FUNCTION_BLOCK ATM_SUB (* Subtracts two TIME values via ATM adapters (F_SUB is ANY_MAGNITUDE, works directly on TIME) *)
  (* Standard: 61499-2; Description: Copyright (c) 2026 HR Agrartechnik GmbH This program and the accompanying materials are made available under the terms of the Eclipse Public License 2.0 which is available at https://www.eclipse.org/legal/epl-2.0/ SPDX-License-Identifier: EPL-2.0 *)
  (* Version 1.0, 2026-08-13, Franz Höpfinger, HR Agrartechnik GmbH, initial API and implementation *)
  PACKAGE adapter::iec61131::arithmetic;
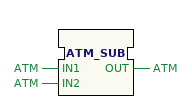
  SOCKETS
    IN1 : adapter::types::unidirectional::ATM; (* First function input *)
    IN2 : adapter::types::unidirectional::ATM; (* Second function input *)
  END_SOCKETS
  PLUGS
    OUT : adapter::types::unidirectional::ATM; (* IN2 subtracted from IN1 *)
  END_PLUGS
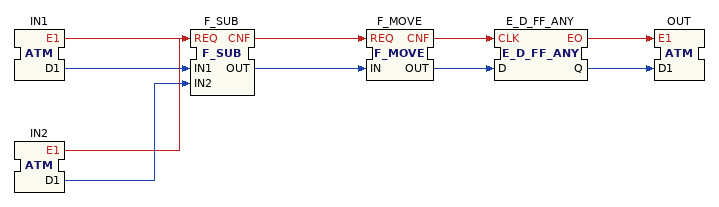
  FBS
    F_SUB : iec61131::arithmetic::F_SUB;
    E_D_FF_ANY : iec61499::events::E_D_FF_ANY;
    F_MOVE : iec61131::selection::F_MOVE; {SET_ATTRIBUTE(DataType, TIME)}
  END_FBS
  EVENT_CONNECTIONS
    IN1.E1 TO F_SUB.REQ;
    IN2.E1 TO F_SUB.REQ;
    E_D_FF_ANY.EO TO OUT.E1;
    F_SUB.CNF TO F_MOVE.REQ;
    F_MOVE.CNF TO E_D_FF_ANY.CLK;
  END_CONNECTIONS
  DATA_CONNECTIONS
    IN1.D1 TO F_SUB.IN1;
    IN2.D1 TO F_SUB.IN2;
    F_SUB.OUT TO F_MOVE.IN;
    E_D_FF_ANY.Q TO OUT.D1;
    F_MOVE.OUT TO E_D_FF_ANY.D;
  END_CONNECTIONS
END_FUNCTION_BLOCK
